RoboDK station: EstacionLEGO_07.rdk

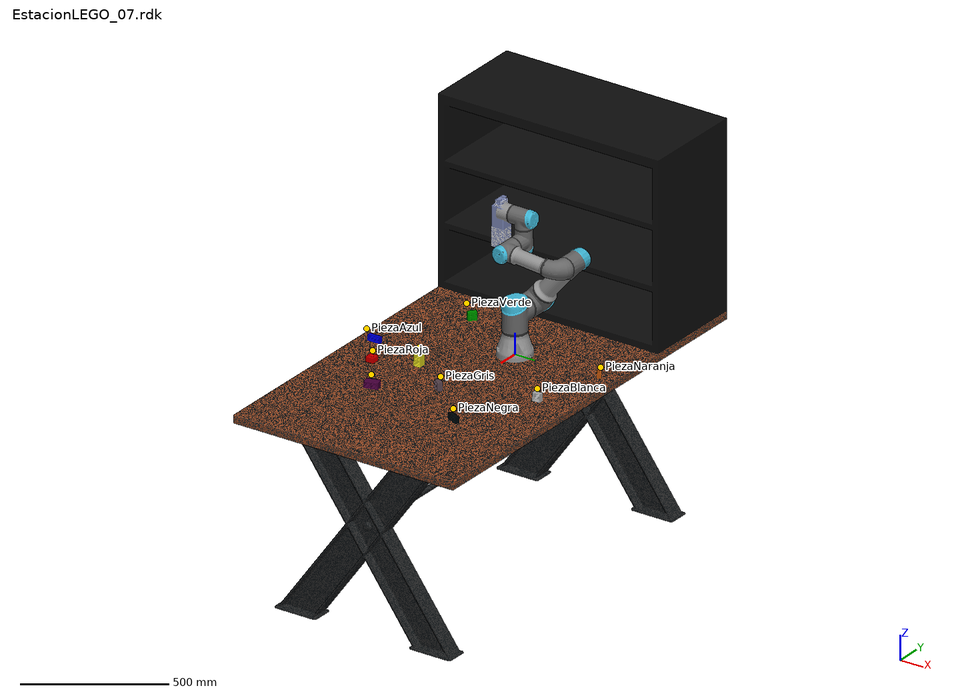
[picture v0: the station drawn from its stored meshes, robots at their saved joint values, targets as dots, program paths as lines]
Station EstacionLEGO_07 (saved by RoboDK 5.4.1). Poses are relative to the parent item; angles as X-Y-Z fixed-axis rotations.
  - frame UR3e Base at (-810.4, -253.58, 719) mm, rotated rx 0 ry 0 rz -90 deg
    - robot UR3e: 6 axes, payload 3 kg, reach 500 mm, repeatability 0.03 mm, weight 11 kg
        modified DH rows (alpha deg, a mm, theta deg, d mm): 0, 0, 0, 151.9; 90, 0, 180, 0; 0, 243.55, 0, 0; 0, 213.2, 0, 131.05; -90, 0, 0, 85.35; 90, 0, 180, 92.1
        joint limits [-360, -360, -360, -360, -360, -360] to [360, 360, 360, 360, 360, 360]; home [0, -90, -90, 0, 90, 0]; saved at [-90, -50, -125, -5, 90, 180]
      - tool RGI-35-14-O-B, TCP at (0, -150, 0) mm, size 50 x 211.5 x 50 mm
    - target PiezaRoja (joint target) at (345.83, -338.28, 58.34) mm, rotated rx 90 ry 0 rz 0 deg; joints [-17.464, -158.43, -55.319, 33.749, 17.464, 180] of UR3e
    - target PiezaVerde (joint target) at (-130.56, -288.31, 58.34) mm, rotated rx 90 ry 0 rz 0 deg; joints [-89.856, -131.778, -129.15, 80.928, 89.856, 180] of UR3e
    - target PiezaAzul (joint target) at (223.29, -448.85, 58.34) mm, rotated rx 90 ry 0 rz 0 deg; joints [-39.815, -157.539, -57.354, 34.893, 39.815, 180] of UR3e
    - target PiezaAmarilla (joint target) at (250.79, -214.14, 65.12) mm, rotated rx 90 ry 0 rz 0 deg; joints [2.077, -133.643, -114.865, 68.508, -2.077, 180] of UR3e
    - target PiezaGris (joint target) at (362.9, -49.71, 48.16) mm, rotated rx 90 ry 0 rz 0 deg; joints [27.681, -148.505, -82.768, 51.273, -27.681, 180] of UR3e
    - target PiezaMorada (joint target) at (484.53, -248.11, 48.16) mm, rotated rx 90 ry 0 rz 63.07 deg; joints [-10.31, -168.442, -35.902, 24.344, 73.382, 180] of UR3e
    - target PiezaBlanca (joint target) at (254.35, 269.63, 48.16) mm, rotated rx 90 ry 0 rz 167.97 deg; joints [63.656, -139.423, -108.46, 67.883, 104.311, 180] of UR3e
    - target PiezaNaranja (joint target) at (-3.2, 347.67, 48.16) mm, rotated rx 90 ry 0 rz -147.27 deg; joints [108.768, -137.356, -115.826, 73.182, 103.961, 180] of UR3e
    - target PiezaNegra (joint target) at (540.57, 128.22, 48.16) mm, rotated rx 90 ry 0 rz 98.85 deg; joints [177.822, -6.275, 24.227, 162.049, -78.968, 180] of UR3e
  - folder Environment
    - object Mesa at (0, 0, -325.07) mm, size 900 x 1600 x 736 mm, geometry from Table IPE.stp
    - object estanteria at (-1319.6, 25, 717.99) mm, size 900 x 400 x 720 mm, geometry from estanteria.stl
  - folder Piezas
    - object 2x2 Green at (-1097.15, -125.08, 718.68) mm, rotated rx 90 ry 0 rz 50.49 deg, size 457 x 44.2 x 285.6 mm
    - object 2x2 Red at (-1134.51, -619.62, 739.15) mm, rotated rx -0.08 ry 0 rz 90 deg, geometry from LEGO_DUPLO_BRICK_2X2.igs
    - object 2x4 Blue at (-1371.17, -448.61, 741.75) mm, size 47.7 x 17.1 x 23.7 mm, geometry from 2x4 lego brick 3001 v6.step
    - object 2x1 Yellow at (-1038.25, -520.57, 769.31) mm, size 50.6 x 37.8 x 25.1 mm, geometry from Duplo 2x1.step
    - object 2x2 Gray at (-871.33, -603.02, 751.72) mm, rotated rx 0 ry 90 rz -129.48 deg, size 31.7 x 31.7 x 23.7 mm, geometry from LEGO_DUPLO_BRICK_2X2.igs
    - object 2x1 Purple at (-1079.48, -754.58, 718.32) mm, rotated rx 0 ry 0 rz 16.1 deg, size 50.6 x 37.8 x 25.1 mm, geometry from Duplo 2x1.step
    - object 2x2 White at (-526.88, -515.12, 752.65) mm, rotated rx 0 ry 90 rz 90 deg, size 31.7 x 31.7 x 23.7 mm, geometry from LEGO_DUPLO_BRICK_2X2.igs
    - object 2x1 Orange at (-485.15, -214.54, 718.7) mm, rotated rx 90 ry 0 rz -54.6 deg, size 30.2 x 22.6 x 15 mm, geometry from Duplo 2x1.step
    - object 2x4 Black at (-798.52, -743.81, 741.77) mm, rotated rx 0 ry 0 rz -24.6 deg, size 47.7 x 17.1 x 23.7 mm, geometry from 2x4 lego brick 3001 v6.step
  - Python program trayectorias (listed below)

--- Python program trayectorias ---
# Type help("robodk.robolink") or help("robodk.robomath") for more information
# Press F5 to run the script
# Documentation: https://robodk.com/doc/en/RoboDK-API.html
# Reference:     https://robodk.com/doc/en/PythonAPI/robodk.html
# Note: It is not required to keep a copy of this file, your Python script is saved with your RDK project
from robodk import robolink    # RoboDK API
from robodk import robomath    # Robot toolbox

# The following 2 lines keep your code compatible with older versions or RoboDK:
from robodk import *      # RoboDK API
from robolink import *    # Robot toolbox

# Start the RoboDK API:
RDK = Robolink()

# Get the robot (first robot found):
robot = RDK.Item('', ITEM_TYPE_ROBOT)

# Getting the reset position -> joints
reset = [-90.00, -50.00, -125.00, -5.00, 90.00, 180.00]

# Getting the target for the two pieces
pRed = RDK.Item('PiezaRoja')
pOrange = RDK.Item('PiezaNaranja')
pYellow = RDK.Item('PiezaAmarilla')
pGreen = RDK.Item('PiezaVerde')
pBlue = RDK.Item('PiezaAzul')
pPurple = RDK.Item('PiezaMorada')
pWhite = RDK.Item('PiezaBlanca')
pBlack = RDK.Item('PiezaNegra')
pGray = RDK.Item('PiezaGris')

# Lista de las posiciones de las piezas en la mesa
piezas = [pRed, pOrange, pYellow, pGreen, pBlue, pPurple, pWhite, pBlack, pGray]

# Getting the final positions for each of the estation cubicles -> Joints
est1 = [-97.00, -110.00, -45.00, -27.00, 97.00, 90.00]
est2 = [-128.00, -68.00, -85.00, -28.00, 128.00, 90.00]
est3 = [-192.00, -80.00, -77.00, -24.00, 158.00, 90.00]
est4 = [-92.00, -119.00, -105.00, 45.00, 97.00, 90.00]
est5 = [-128.00, -85.00, -152.00, 57.00, 128.00, 90.00]
est6 = [-192.00, -92.00, -135.00, 45.00, 158.00, 90.00]
est7 = [-95.00, -145.00, -70.00, -143.00, 50.00, 90.00]
est8 = [-97.00, -125.00, -125.00, -115.00, 90.00, 90.00]
est9 = [-180.00, -119.00, -144.00, -99.00, 5.00, 90.00]

# Antes tenemos los targets a donde queremos mover el robot
# las estaciones de posicion finales
estaciones = [est1, est2, est3, est4, est5, est6, est7, est8, est9]

# Go to reset position:
robot.setJoints(reset)

# Movimiento
numEstaciones = 9
for i in range(numEstaciones):
    robot.MoveJ(piezas[i])
    robot.MoveJ(estaciones[i])
    robot.MoveJ(reset)
    robot.Pause(3000)


# Trigger a program call at the end of the movement
robot.RunInstruction('Program_Done')
